FUNCTION_BLOCK DSCYL_PRXY (* Proxy for a Remote Double-Stroke Cylinder *)
  (* Standard: 61499-1 *)
  (* Version 0.0, 2004-09-26, JHC, Rockwell Automation, Adapted from DSCYL_MDL1. *)
  (* Compiler header: package fb.rt.mach; import fb.rt.net.*; *)
  (* Compiler Java Sun JDK 1.4.2 *)
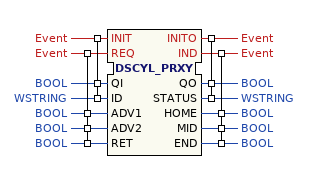
  EVENT_INPUT
    INIT WITH QI, ID; (* Initialize Client/Server Connection *)
    REQ WITH ADV1, ADV2, RET; (* Send Actuator Data *)
  END_EVENT
  EVENT_OUTPUT
    INITO WITH QO, STATUS; (* INIT Acknowledgment *)
    IND WITH HOME, MID, END; (* Sensor Change Indication *)
  END_EVENT
  VAR_INPUT
    QI : BOOL; (* Event Input Qualifier *)
    ID : WSTRING; (* Connection Identifier *)
    ADV1 : BOOL; (* ADVANCE Cyl#1 *)
    ADV2 : BOOL; (* ADVANCE Cyl#2 *)
    RET : BOOL; (* RETRACT Both Cylinders *)
  END_VAR
  VAR_OUTPUT
    QO : BOOL; (* Event Output Qualifier *)
    STATUS : WSTRING; (* Service Status *)
    HOME : BOOL; (* Both cylinders HOME *)
    MID : BOOL; (* CYL1 at END,CYL2 HOME *)
    END : BOOL; (* Both cylinders at END *)
  END_VAR
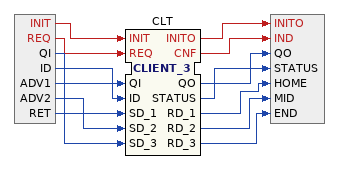
  FBS
    CLT : CLIENT_3;
  END_FBS
  EVENT_CONNECTIONS
    INIT TO CLT.INIT;
    CLT.INITO TO INITO;
    CLT.CNF TO IND;
    REQ TO CLT.REQ;
  END_CONNECTIONS
  DATA_CONNECTIONS
    QI TO CLT.QI;
    CLT.QO TO QO;
    ID TO CLT.ID;
    CLT.STATUS TO STATUS;
    ADV1 TO CLT.SD_1;
    ADV2 TO CLT.SD_2;
    RET TO CLT.SD_3;
    CLT.RD_1 TO HOME;
    CLT.RD_2 TO MID;
    CLT.RD_3 TO END;
  END_CONNECTIONS
END_FUNCTION_BLOCK
